# EPICS StreamDevice protocol: protocols/acq43x.proto
Terminator = LF;
ExtraInput = Ignore;

setNacc {
	out "nacc %d";
	in;
}

getNacc {
	out "nacc";
	in "%d,%*d";
	@replytimeout {
		disconnect;
		wait 2000;
		connect 1000;
	}
}

setRtmTranslen {
	out "rtm_translen %d";
	in;
}

getRtmTranslen {
	out "rtm_translen";
	in "%d";
}

getDiv {
	in "%*d,%d";
}

setHiResMode {
	out "hi_res_mode %d";
	in;
}

getHiResMode {
	out "hi_res_mode";
	in "%d";
}
